{attribute 'GeneratedUsingTerminal: CU2508-0000-0016'}
{attribute addProperty BoxType "CU2508-0000-0016"}
{attribute addProperty Description "CU2508 Configuration Port"}
{attribute addProperty Physics "YY"}
{attribute addProperty Id "InfoDataAT %I*InfoData_32EB74EA10"}
{attribute addProperty CRC "4004708084"}
{attribute addProperty Size "10"}
TYPE CU2508_EEB2FEF4 EXTENDS EtcSlaveBoxBase_77A0E4A7 :
STRUCT
	{attribute addProperty Name "InfoData"}
	InfoData : InfoData_32EB74EA;
END_STRUCT
END_TYPE

(* stored: Version 1.2.0.0, ProductVersion 3.1.4024.11
   DUT CU2508_EEB2FEF4: Id {785a8af1-231d-4f78-b90f-44be77c6c458} *)
